Staubli VAL3: whichObjectUsed.pgx

public program whichObjectUsed(num& x_nIdxInUse[])
begin
  // This checks if the index pointed by nIdxPull activated
  // It is activated when getNextID has been called once and
  // there is an object in the queue
  //
  // Input param
  //  none
  //
  // Output param
  //  x_nIdxInUse : Index in the queue that is currently activated
  //
  // Created 25-01-06                                   C.CURRIVAND
  //----------------------------------------------------------------
  //
  x_nIdxInUse=sel(nNumbOfUser[nIdxPull]>0,nIdxPull,-1)
end
